// TIA Portal V20 export
FUNCTION_BLOCK "Sequence_1_StackNgBox"   // FB32864, LAD
TITLE = Sequence
// Sequence template programmend in ladder logic
// stored: IsIECCheckEnabled true, MemoryReserve 100, Namespace Unit1.Em12, SetENOAutomatically true
   VAR_INPUT
      unitStatus { ExternalAccessible := 'False'; ExternalVisible := 'False'; ExternalWritable := 'False'} : "LAF_typeUnitStatus";   // Current unit status o be used in this EM
   END_VAR
   VAR
      instSequenceLADControl { ExternalAccessible := 'False'; ExternalVisible := 'False'; ExternalWritable := 'False'} : "LAF_ControlLadSequence";
      instSequenceLADStatus { ExternalAccessible := 'False'; ExternalVisible := 'False'; ExternalWritable := 'False'} : "LAF_StatusLadSequence";
      statTonTime { ExternalAccessible := 'False'; ExternalVisible := 'False'; ExternalWritable := 'False'} : Array[0..9999] of TON_TIME;
      NoDataCheck { S7_SetPoint := 'True'} : "LER_typePartData";
   END_VAR
   VAR_TEMP
      tempCustomerAction : Bool;   // Placeholder for possible actions
      tempDo_nothing_and_wait_for_init : Bool;   // Placeholder for doing nothing
      tempSafeStateCondition : Bool;   // Temp Condition for the equipment module to be in a safe state
   END_VAR
   VAR CONSTANT
      delayTime : Time := T#500ms;
      STEP_IDLE : DInt := 1;
      JOB_1_STEP_01 : DInt := 101;
      JOB_1_STEP_10 : DInt := 110;
      JOB_1_STEP_20 : DInt := 120;
      JOB_1_STEP_30 : DInt := 130;
      JOB_1_STEP_40 : DInt := 140;
      JOB_1_STEP_50 : DInt := 150;
      JOB_1_STEP_60 : DInt := 160;
      JOB_1_STEP_70 : DInt := 170;
      JOB_1_STEP_80 : DInt := 180;
      JOB_1_STEP_90 : DInt := 190;
      JOB_2_STEP_01 : DInt := 201;
      JOB_2_STEP_10 : DInt := 210;
      JOB_2_STEP_20 : DInt := 220;
      JOB_2_STEP_30 : DInt := 230;
      JOB_2_STEP_31 : DInt := 231;
      JOB_2_STEP_40 : DInt := 240;
      JOB_2_STEP_50 : DInt := 250;
      JOB_2_STEP_60 : DInt := 260;
      JOB_2_STEP_70 : DInt := 270;
      JOB_2_STEP_80 : DInt := 280;
      JOB_2_STEP_90 : DInt := 290;
      JOB_3_STEP_01 : DInt := 301;
      JOB_3_STEP_10 : DInt := 310;
      JOB_3_STEP_20 : DInt := 320;
      JOB_3_STEP_30 : DInt := 330;
      JOB_3_STEP_40 : DInt := 340;
      JOB_3_STEP_50 : DInt := 350;
      JOB_3_STEP_60 : DInt := 360;
      JOB_3_STEP_70 : DInt := 370;
      JOB_3_STEP_80 : DInt := 380;
      JOB_3_STEP_90 : DInt := 390;
      STEP_IMMEDIATE_STOP : DInt := 9001;   // Step executed when an immediate stop command is triggered for the sequence (i.e. when unit is in state aborting)
   END_VAR
   VAR_TEMP   // added for the SCL form of the ladder/FBD networks
      _w1 : Bool;
      _w2 : Bool;
   END_VAR
BEGIN

REGION Network 1: BLOCK INFO HEADER
   // (company) / (C) Copyright (year)
   // ---------------------------------------------------------------------------------
   // Title:                             (Title of this block)
   // Comment/Function: (that is implemented in the block)
   // Library/Family:           (that the source is dedicated to)
   // Author:                        (department / person in charge / contact)
   // Target System:          (test system with FW version)
   // Engineering:              TIA Portal (SW version)
   // Restrictions:               (OB types, etc.)
   // Requirements:           (hardware, technological package, etc.)
   // ---------------------------------------------------------------------------------
   // Change log table:
   // Version          | Date             | Signature      | Expert in charge  | Changes applied ------------------------|----------------------|-------------------------|--------------------------------|-----------------------
   // 001.000.000 | yyyy-mm-dd | 0x00000000 | (name of expert) | First released version
END_REGION

REGION Network 2 (SCL): DESCRIPTION
   // This is a template block provided by the Automation Framework. It can be used to create an own project.
   // The Block Info Header is prepared to put in your own data.
   // Description of the block could be added here and the docu created by Code2Docu.
   // 1. Home 동작 시 NG box 감지 유무에 따라 Lock, Unlock이 되면 박스의 위치가 정확하지 않을 때는 불합리하므로 작업자의 수동 작업 필요.
END_REGION

REGION Network 3: ********************* CONTROL *************************
END_REGION

REGION Network 4: Sequence Control ("Enter your Sequins number here")
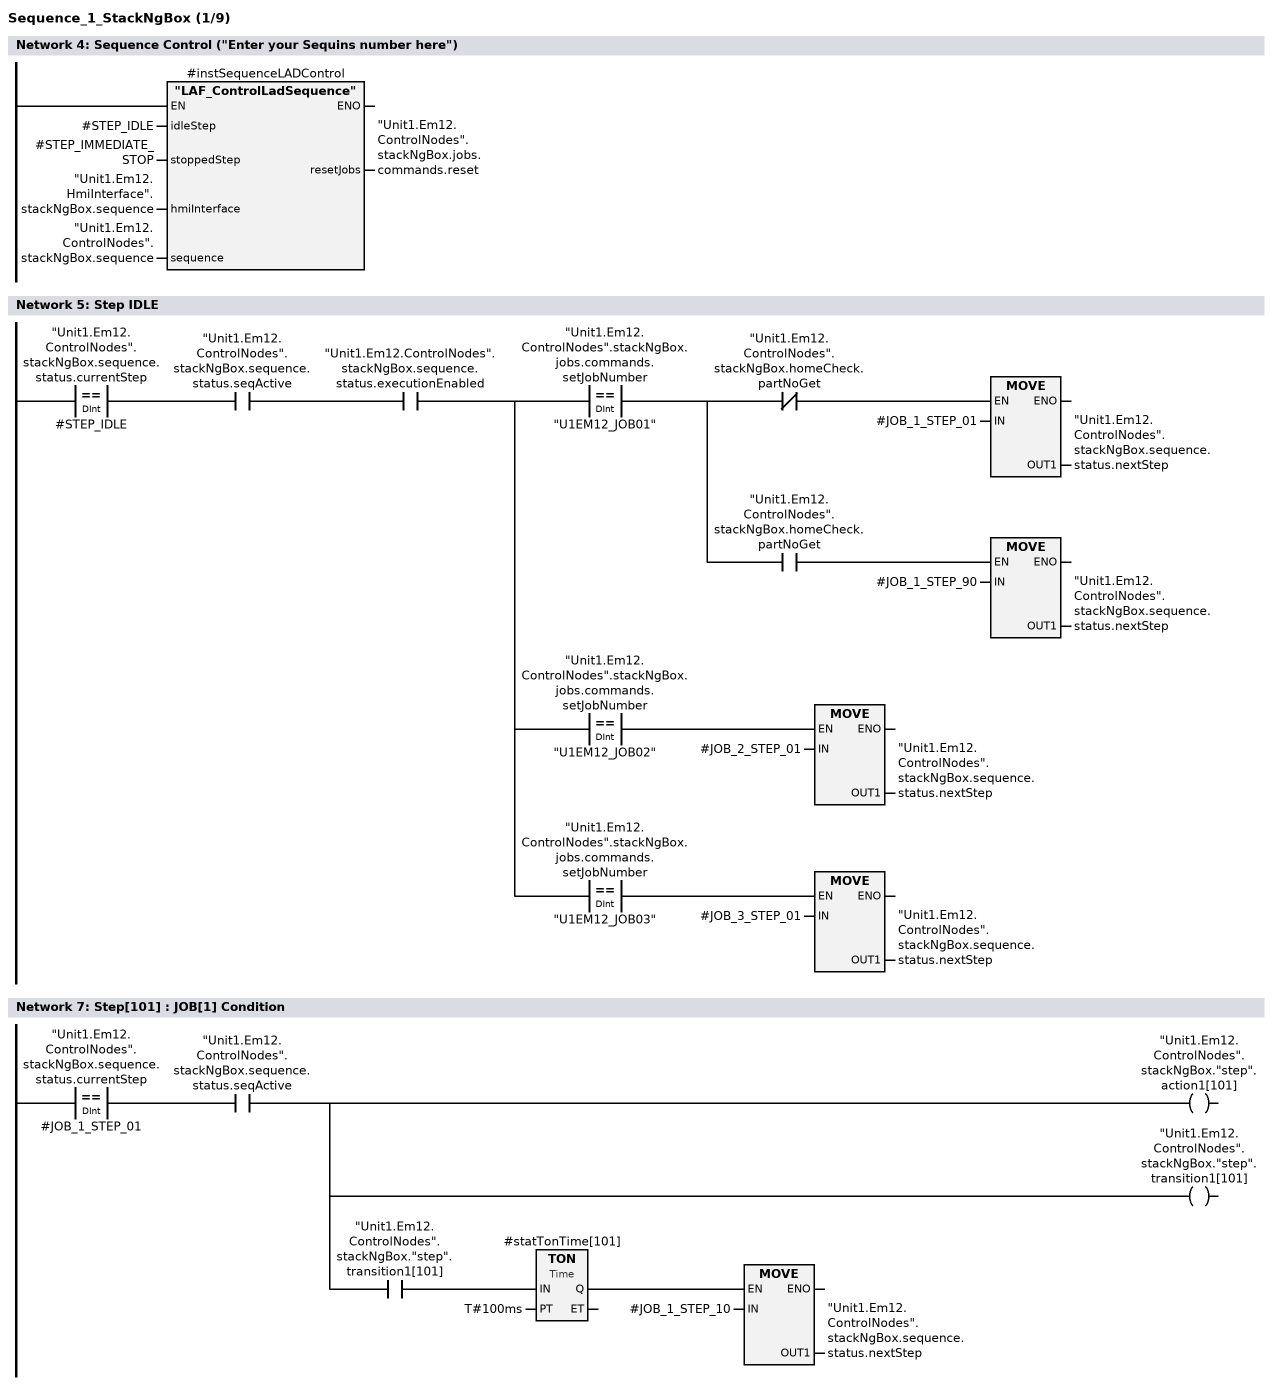
   RUNG wire#powerrail
      #instSequenceLADControl(idleStep := #STEP_IDLE, stoppedStep := #STEP_IMMEDIATE_STOP, hmiInterface := "Unit1.Em12.HmiInterface".stackNgBox.sequence, sequence := "Unit1.Em12.ControlNodes".stackNgBox.sequence, resetJobs => "Unit1.Em12.ControlNodes".stackNgBox.jobs.commands.reset)
   END_RUNG
   // the same network as SCL:
   #instSequenceLADControl(idleStep := #STEP_IDLE,   // "LAF_ControlLadSequence"
                           stoppedStep := #STEP_IMMEDIATE_STOP,
                           hmiInterface := "Unit1.Em12.HmiInterface".stackNgBox.sequence,
                           sequence := "Unit1.Em12.ControlNodes".stackNgBox.sequence,
                           resetJobs => "Unit1.Em12.ControlNodes".stackNgBox.jobs.commands.reset);
END_REGION

REGION Network 5: Step IDLE
   RUNG wire#powerrail
      { S7_Templates := "SrcType := DInt" } EQ_Contact(in1 := "Unit1.Em12.ControlNodes".stackNgBox.sequence.status.currentStep, in2 := #STEP_IDLE)
      Contact( "Unit1.Em12.ControlNodes".stackNgBox.sequence.status.seqActive )
      Contact( "Unit1.Em12.ControlNodes".stackNgBox.sequence.status.executionEnabled )
      wire#w1
      { S7_Templates := "SrcType := DInt" } EQ_Contact(in1 := "Unit1.Em12.ControlNodes".stackNgBox.jobs.commands.setJobNumber, in2 := "U1EM12_JOB01")
      wire#w2
      I_Contact( "Unit1.Em12.ControlNodes".stackNgBox.homeCheck.partNoGet )
      Move(in := #JOB_1_STEP_01, out1 => "Unit1.Em12.ControlNodes".stackNgBox.sequence.status.nextStep)
   END_RUNG
   RUNG wire#w2
      Contact( "Unit1.Em12.ControlNodes".stackNgBox.homeCheck.partNoGet )
      Move(in := #JOB_1_STEP_90, out1 => "Unit1.Em12.ControlNodes".stackNgBox.sequence.status.nextStep)
   END_RUNG
   RUNG wire#w1
      { S7_Templates := "SrcType := DInt" } EQ_Contact(in1 := "Unit1.Em12.ControlNodes".stackNgBox.jobs.commands.setJobNumber, in2 := "U1EM12_JOB02")
      Move(in := #JOB_2_STEP_01, out1 => "Unit1.Em12.ControlNodes".stackNgBox.sequence.status.nextStep)
   END_RUNG
   RUNG wire#w1
      { S7_Templates := "SrcType := DInt" } EQ_Contact(in1 := "Unit1.Em12.ControlNodes".stackNgBox.jobs.commands.setJobNumber, in2 := "U1EM12_JOB03")
      Move(in := #JOB_3_STEP_01, out1 => "Unit1.Em12.ControlNodes".stackNgBox.sequence.status.nextStep)
   END_RUNG
   // the same network as SCL:
   #_w1 := ("Unit1.Em12.ControlNodes".stackNgBox.sequence.status.currentStep = #STEP_IDLE) AND "Unit1.Em12.ControlNodes".stackNgBox.sequence.status.seqActive AND "Unit1.Em12.ControlNodes".stackNgBox.sequence.status.executionEnabled;
   #_w2 := #_w1 AND ("Unit1.Em12.ControlNodes".stackNgBox.jobs.commands.setJobNumber = "U1EM12_JOB01");
   IF #_w2 AND NOT "Unit1.Em12.ControlNodes".stackNgBox.homeCheck.partNoGet THEN
       "Unit1.Em12.ControlNodes".stackNgBox.sequence.status.nextStep := #JOB_1_STEP_01;
   END_IF;
   IF #_w2 AND "Unit1.Em12.ControlNodes".stackNgBox.homeCheck.partNoGet THEN
       "Unit1.Em12.ControlNodes".stackNgBox.sequence.status.nextStep := #JOB_1_STEP_90;
   END_IF;
   IF #_w1 AND ("Unit1.Em12.ControlNodes".stackNgBox.jobs.commands.setJobNumber = "U1EM12_JOB02") THEN
       "Unit1.Em12.ControlNodes".stackNgBox.sequence.status.nextStep := #JOB_2_STEP_01;
   END_IF;
   IF #_w1 AND ("Unit1.Em12.ControlNodes".stackNgBox.jobs.commands.setJobNumber = "U1EM12_JOB03") THEN
       "Unit1.Em12.ControlNodes".stackNgBox.sequence.status.nextStep := #JOB_3_STEP_01;
   END_IF;
END_REGION

REGION Network 6: *************** JOB[1] EM HOMING ************************
END_REGION

REGION Network 7: Step[101] : JOB[1] Condition
   RUNG wire#powerrail
      { S7_Templates := "SrcType := DInt" } EQ_Contact(in1 := "Unit1.Em12.ControlNodes".stackNgBox.sequence.status.currentStep, in2 := #JOB_1_STEP_01)
      Contact( "Unit1.Em12.ControlNodes".stackNgBox.sequence.status.seqActive )
      wire#w1
      Coil( "Unit1.Em12.ControlNodes".stackNgBox."step".action1[101] )
   END_RUNG
   RUNG wire#w1
      Coil( "Unit1.Em12.ControlNodes".stackNgBox."step".transition1[101] )
   END_RUNG
   RUNG wire#w1
      Contact( "Unit1.Em12.ControlNodes".stackNgBox."step".transition1[101] )
      { S7_Templates := "time_type := Time" } #statTonTime[101].TON(pt := T#100ms, et =>)
      Move(in := #JOB_1_STEP_10, out1 => "Unit1.Em12.ControlNodes".stackNgBox.sequence.status.nextStep)
   END_RUNG
   // the same network as SCL:
   "Unit1.Em12.ControlNodes".stackNgBox."step".action1[101] := ("Unit1.Em12.ControlNodes".stackNgBox.sequence.status.currentStep = #JOB_1_STEP_01) AND "Unit1.Em12.ControlNodes".stackNgBox.sequence.status.seqActive;
   "Unit1.Em12.ControlNodes".stackNgBox."step".transition1[101] := ("Unit1.Em12.ControlNodes".stackNgBox.sequence.status.currentStep = #JOB_1_STEP_01) AND "Unit1.Em12.ControlNodes".stackNgBox.sequence.status.seqActive;
   #statTonTime[101].TON(IN := ("Unit1.Em12.ControlNodes".stackNgBox.sequence.status.currentStep = #JOB_1_STEP_01) AND "Unit1.Em12.ControlNodes".stackNgBox.sequence.status.seqActive AND "Unit1.Em12.ControlNodes".stackNgBox."step".transition1[101],
                         PT := T#100ms);
   IF #statTonTime[101].Q THEN
       "Unit1.Em12.ControlNodes".stackNgBox.sequence.status.nextStep := #JOB_1_STEP_10;
   END_IF;
END_REGION

REGION Network 8: Step[110] : Clamp Z Up
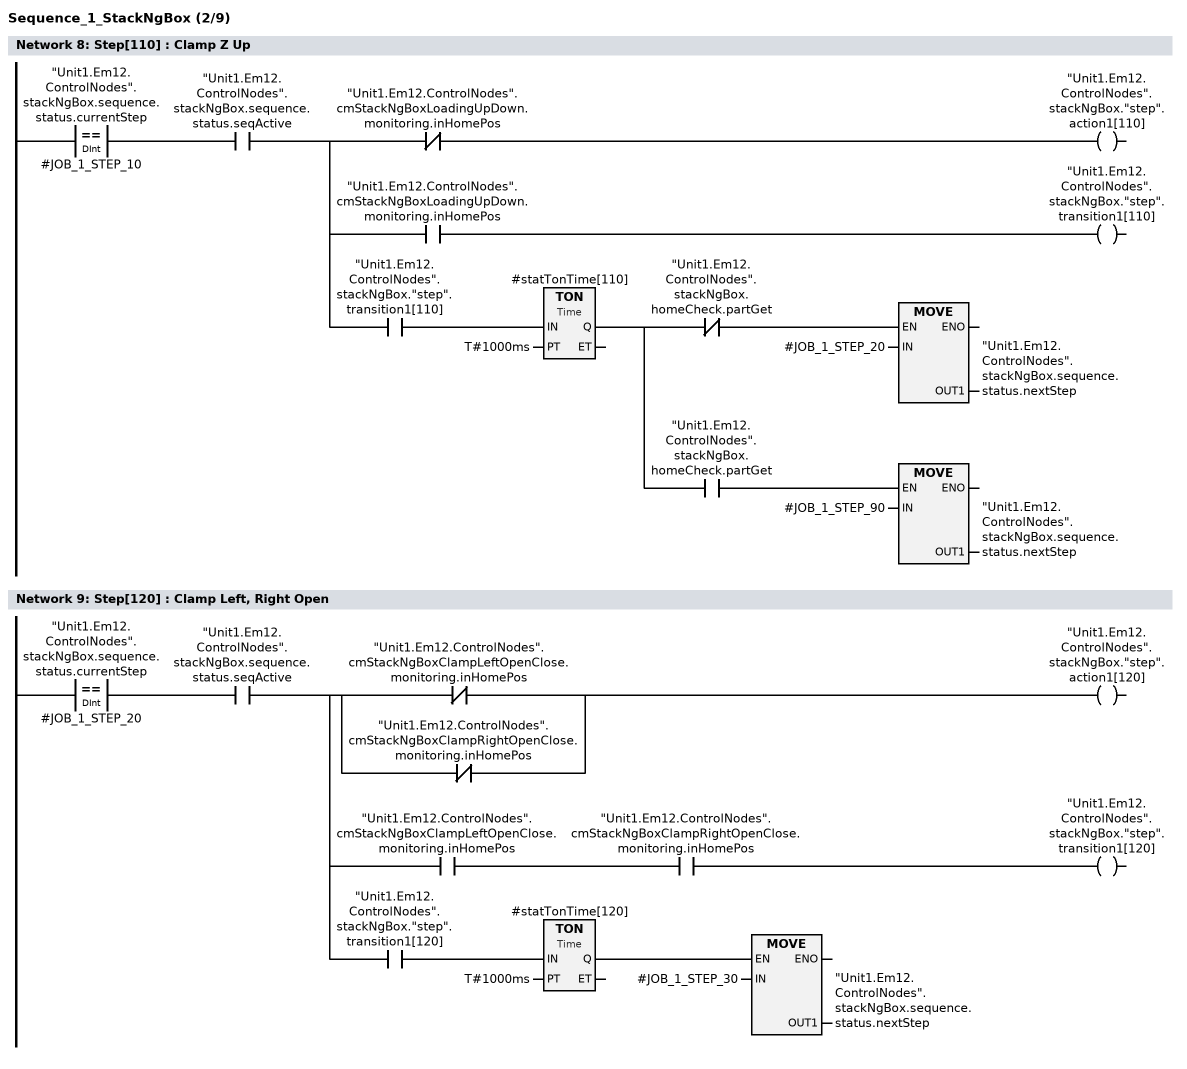
   RUNG wire#powerrail
      { S7_Templates := "SrcType := DInt" } EQ_Contact(in1 := "Unit1.Em12.ControlNodes".stackNgBox.sequence.status.currentStep, in2 := #JOB_1_STEP_10)
      Contact( "Unit1.Em12.ControlNodes".stackNgBox.sequence.status.seqActive )
      wire#w1
      I_Contact( "Unit1.Em12.ControlNodes".cmStackNgBoxLoadingUpDown.monitoring.inHomePos )
      Coil( "Unit1.Em12.ControlNodes".stackNgBox."step".action1[110] )
   END_RUNG
   RUNG wire#w1
      Contact( "Unit1.Em12.ControlNodes".cmStackNgBoxLoadingUpDown.monitoring.inHomePos )
      Coil( "Unit1.Em12.ControlNodes".stackNgBox."step".transition1[110] )
   END_RUNG
   RUNG wire#w1
      Contact( "Unit1.Em12.ControlNodes".stackNgBox."step".transition1[110] )
      { S7_Templates := "time_type := Time" } #statTonTime[110].TON(pt := T#1000ms, et =>)
      wire#w2
      I_Contact( "Unit1.Em12.ControlNodes".stackNgBox.homeCheck.partGet )
      Move(in := #JOB_1_STEP_20, out1 => "Unit1.Em12.ControlNodes".stackNgBox.sequence.status.nextStep)
   END_RUNG
   RUNG wire#w2
      Contact( "Unit1.Em12.ControlNodes".stackNgBox.homeCheck.partGet )
      Move(in := #JOB_1_STEP_90, out1 => "Unit1.Em12.ControlNodes".stackNgBox.sequence.status.nextStep)
   END_RUNG
   // the same network as SCL:
   #_w1 := ("Unit1.Em12.ControlNodes".stackNgBox.sequence.status.currentStep = #JOB_1_STEP_10) AND "Unit1.Em12.ControlNodes".stackNgBox.sequence.status.seqActive;
   "Unit1.Em12.ControlNodes".stackNgBox."step".action1[110] := #_w1 AND NOT "Unit1.Em12.ControlNodes".cmStackNgBoxLoadingUpDown.monitoring.inHomePos;
   "Unit1.Em12.ControlNodes".stackNgBox."step".transition1[110] := #_w1 AND "Unit1.Em12.ControlNodes".cmStackNgBoxLoadingUpDown.monitoring.inHomePos;
   #statTonTime[110].TON(IN := #_w1 AND "Unit1.Em12.ControlNodes".stackNgBox."step".transition1[110],
                         PT := T#1000ms);
   IF #statTonTime[110].Q AND NOT "Unit1.Em12.ControlNodes".stackNgBox.homeCheck.partGet THEN
       "Unit1.Em12.ControlNodes".stackNgBox.sequence.status.nextStep := #JOB_1_STEP_20;
   END_IF;
   IF #statTonTime[110].Q AND "Unit1.Em12.ControlNodes".stackNgBox.homeCheck.partGet THEN
       "Unit1.Em12.ControlNodes".stackNgBox.sequence.status.nextStep := #JOB_1_STEP_90;
   END_IF;
END_REGION

REGION Network 9: Step[120] : Clamp Left, Right Open
   RUNG wire#powerrail
      { S7_Templates := "SrcType := DInt" } EQ_Contact(in1 := "Unit1.Em12.ControlNodes".stackNgBox.sequence.status.currentStep, in2 := #JOB_1_STEP_20)
      Contact( "Unit1.Em12.ControlNodes".stackNgBox.sequence.status.seqActive )
      wire#w1
      I_Contact( "Unit1.Em12.ControlNodes".cmStackNgBoxClampLeftOpenClose.monitoring.inHomePos )
      wire#w2
      Coil( "Unit1.Em12.ControlNodes".stackNgBox."step".action1[120] )
   END_RUNG
   RUNG wire#w1
      I_Contact( "Unit1.Em12.ControlNodes".cmStackNgBoxClampRightOpenClose.monitoring.inHomePos )
   END_RUNG wire#w2
   RUNG wire#w1
      Contact( "Unit1.Em12.ControlNodes".cmStackNgBoxClampLeftOpenClose.monitoring.inHomePos )
      Contact( "Unit1.Em12.ControlNodes".cmStackNgBoxClampRightOpenClose.monitoring.inHomePos )
      Coil( "Unit1.Em12.ControlNodes".stackNgBox."step".transition1[120] )
   END_RUNG
   RUNG wire#w1
      Contact( "Unit1.Em12.ControlNodes".stackNgBox."step".transition1[120] )
      { S7_Templates := "time_type := Time" } #statTonTime[120].TON(pt := T#1000ms, et =>)
      Move(in := #JOB_1_STEP_30, out1 => "Unit1.Em12.ControlNodes".stackNgBox.sequence.status.nextStep)
   END_RUNG
   // the same network as SCL:
   #_w1 := ("Unit1.Em12.ControlNodes".stackNgBox.sequence.status.currentStep = #JOB_1_STEP_20) AND "Unit1.Em12.ControlNodes".stackNgBox.sequence.status.seqActive;
   "Unit1.Em12.ControlNodes".stackNgBox."step".action1[120] := #_w1 AND (NOT "Unit1.Em12.ControlNodes".cmStackNgBoxClampLeftOpenClose.monitoring.inHomePos OR NOT "Unit1.Em12.ControlNodes".cmStackNgBoxClampRightOpenClose.monitoring.inHomePos);
   "Unit1.Em12.ControlNodes".stackNgBox."step".transition1[120] := #_w1 AND "Unit1.Em12.ControlNodes".cmStackNgBoxClampLeftOpenClose.monitoring.inHomePos AND "Unit1.Em12.ControlNodes".cmStackNgBoxClampRightOpenClose.monitoring.inHomePos;
   #statTonTime[120].TON(IN := #_w1 AND "Unit1.Em12.ControlNodes".stackNgBox."step".transition1[120],
                         PT := T#1000ms);
   IF #statTonTime[120].Q THEN
       "Unit1.Em12.ControlNodes".stackNgBox.sequence.status.nextStep := #JOB_1_STEP_30;
   END_IF;
END_REGION

REGION Network 10: Step[130] : Clamp Mover Open
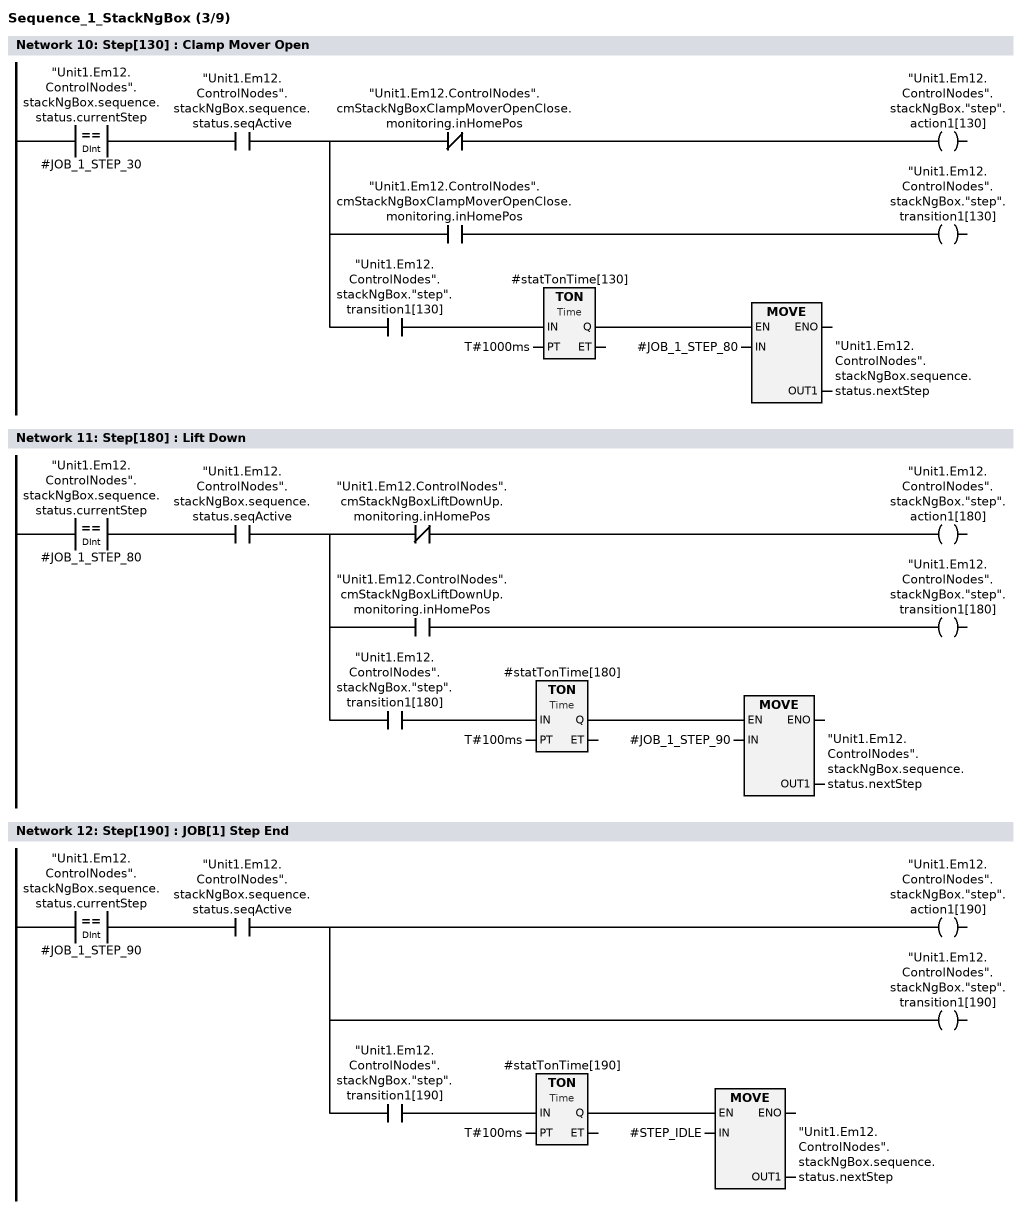
   RUNG wire#powerrail
      { S7_Templates := "SrcType := DInt" } EQ_Contact(in1 := "Unit1.Em12.ControlNodes".stackNgBox.sequence.status.currentStep, in2 := #JOB_1_STEP_30)
      Contact( "Unit1.Em12.ControlNodes".stackNgBox.sequence.status.seqActive )
      wire#w1
      I_Contact( "Unit1.Em12.ControlNodes".cmStackNgBoxClampMoverOpenClose.monitoring.inHomePos )
      Coil( "Unit1.Em12.ControlNodes".stackNgBox."step".action1[130] )
   END_RUNG
   RUNG wire#w1
      Contact( "Unit1.Em12.ControlNodes".cmStackNgBoxClampMoverOpenClose.monitoring.inHomePos )
      Coil( "Unit1.Em12.ControlNodes".stackNgBox."step".transition1[130] )
   END_RUNG
   RUNG wire#w1
      Contact( "Unit1.Em12.ControlNodes".stackNgBox."step".transition1[130] )
      { S7_Templates := "time_type := Time" } #statTonTime[130].TON(pt := T#1000ms, et =>)
      Move(in := #JOB_1_STEP_80, out1 => "Unit1.Em12.ControlNodes".stackNgBox.sequence.status.nextStep)
   END_RUNG
   // the same network as SCL:
   #_w1 := ("Unit1.Em12.ControlNodes".stackNgBox.sequence.status.currentStep = #JOB_1_STEP_30) AND "Unit1.Em12.ControlNodes".stackNgBox.sequence.status.seqActive;
   "Unit1.Em12.ControlNodes".stackNgBox."step".action1[130] := #_w1 AND NOT "Unit1.Em12.ControlNodes".cmStackNgBoxClampMoverOpenClose.monitoring.inHomePos;
   "Unit1.Em12.ControlNodes".stackNgBox."step".transition1[130] := #_w1 AND "Unit1.Em12.ControlNodes".cmStackNgBoxClampMoverOpenClose.monitoring.inHomePos;
   #statTonTime[130].TON(IN := #_w1 AND "Unit1.Em12.ControlNodes".stackNgBox."step".transition1[130],
                         PT := T#1000ms);
   IF #statTonTime[130].Q THEN
       "Unit1.Em12.ControlNodes".stackNgBox.sequence.status.nextStep := #JOB_1_STEP_80;
   END_IF;
END_REGION

REGION Network 11: Step[180] : Lift Down
   RUNG wire#powerrail
      { S7_Templates := "SrcType := DInt" } EQ_Contact(in1 := "Unit1.Em12.ControlNodes".stackNgBox.sequence.status.currentStep, in2 := #JOB_1_STEP_80)
      Contact( "Unit1.Em12.ControlNodes".stackNgBox.sequence.status.seqActive )
      wire#w1
      I_Contact( "Unit1.Em12.ControlNodes".cmStackNgBoxLiftDownUp.monitoring.inHomePos )
      Coil( "Unit1.Em12.ControlNodes".stackNgBox."step".action1[180] )
   END_RUNG
   RUNG wire#w1
      Contact( "Unit1.Em12.ControlNodes".cmStackNgBoxLiftDownUp.monitoring.inHomePos )
      Coil( "Unit1.Em12.ControlNodes".stackNgBox."step".transition1[180] )
   END_RUNG
   RUNG wire#w1
      Contact( "Unit1.Em12.ControlNodes".stackNgBox."step".transition1[180] )
      { S7_Templates := "time_type := Time" } #statTonTime[180].TON(pt := T#100ms, et =>)
      Move(in := #JOB_1_STEP_90, out1 => "Unit1.Em12.ControlNodes".stackNgBox.sequence.status.nextStep)
   END_RUNG
   // the same network as SCL:
   #_w1 := ("Unit1.Em12.ControlNodes".stackNgBox.sequence.status.currentStep = #JOB_1_STEP_80) AND "Unit1.Em12.ControlNodes".stackNgBox.sequence.status.seqActive;
   "Unit1.Em12.ControlNodes".stackNgBox."step".action1[180] := #_w1 AND NOT "Unit1.Em12.ControlNodes".cmStackNgBoxLiftDownUp.monitoring.inHomePos;
   "Unit1.Em12.ControlNodes".stackNgBox."step".transition1[180] := #_w1 AND "Unit1.Em12.ControlNodes".cmStackNgBoxLiftDownUp.monitoring.inHomePos;
   #statTonTime[180].TON(IN := #_w1 AND "Unit1.Em12.ControlNodes".stackNgBox."step".transition1[180],
                         PT := T#100ms);
   IF #statTonTime[180].Q THEN
       "Unit1.Em12.ControlNodes".stackNgBox.sequence.status.nextStep := #JOB_1_STEP_90;
   END_IF;
END_REGION

REGION Network 12: Step[190] : JOB[1] Step End
   RUNG wire#powerrail
      { S7_Templates := "SrcType := DInt" } EQ_Contact(in1 := "Unit1.Em12.ControlNodes".stackNgBox.sequence.status.currentStep, in2 := #JOB_1_STEP_90)
      Contact( "Unit1.Em12.ControlNodes".stackNgBox.sequence.status.seqActive )
      wire#w1
      Coil( "Unit1.Em12.ControlNodes".stackNgBox."step".action1[190] )
   END_RUNG
   RUNG wire#w1
      Coil( "Unit1.Em12.ControlNodes".stackNgBox."step".transition1[190] )
   END_RUNG
   RUNG wire#w1
      Contact( "Unit1.Em12.ControlNodes".stackNgBox."step".transition1[190] )
      { S7_Templates := "time_type := Time" } #statTonTime[190].TON(pt := T#100ms, et =>)
      Move(in := #STEP_IDLE, out1 => "Unit1.Em12.ControlNodes".stackNgBox.sequence.status.nextStep)
   END_RUNG
   // the same network as SCL:
   "Unit1.Em12.ControlNodes".stackNgBox."step".action1[190] := ("Unit1.Em12.ControlNodes".stackNgBox.sequence.status.currentStep = #JOB_1_STEP_90) AND "Unit1.Em12.ControlNodes".stackNgBox.sequence.status.seqActive;
   "Unit1.Em12.ControlNodes".stackNgBox."step".transition1[190] := ("Unit1.Em12.ControlNodes".stackNgBox.sequence.status.currentStep = #JOB_1_STEP_90) AND "Unit1.Em12.ControlNodes".stackNgBox.sequence.status.seqActive;
   #statTonTime[190].TON(IN := ("Unit1.Em12.ControlNodes".stackNgBox.sequence.status.currentStep = #JOB_1_STEP_90) AND "Unit1.Em12.ControlNodes".stackNgBox.sequence.status.seqActive AND "Unit1.Em12.ControlNodes".stackNgBox."step".transition1[190],
                         PT := T#100ms);
   IF #statTonTime[190].Q THEN
       "Unit1.Em12.ControlNodes".stackNgBox.sequence.status.nextStep := #STEP_IDLE;
   END_IF;
END_REGION

REGION Network 13: *************** JOB[2] JR GET=AUTO **********************
END_REGION

REGION Network 14: Step[201] : JOB[2] Condition
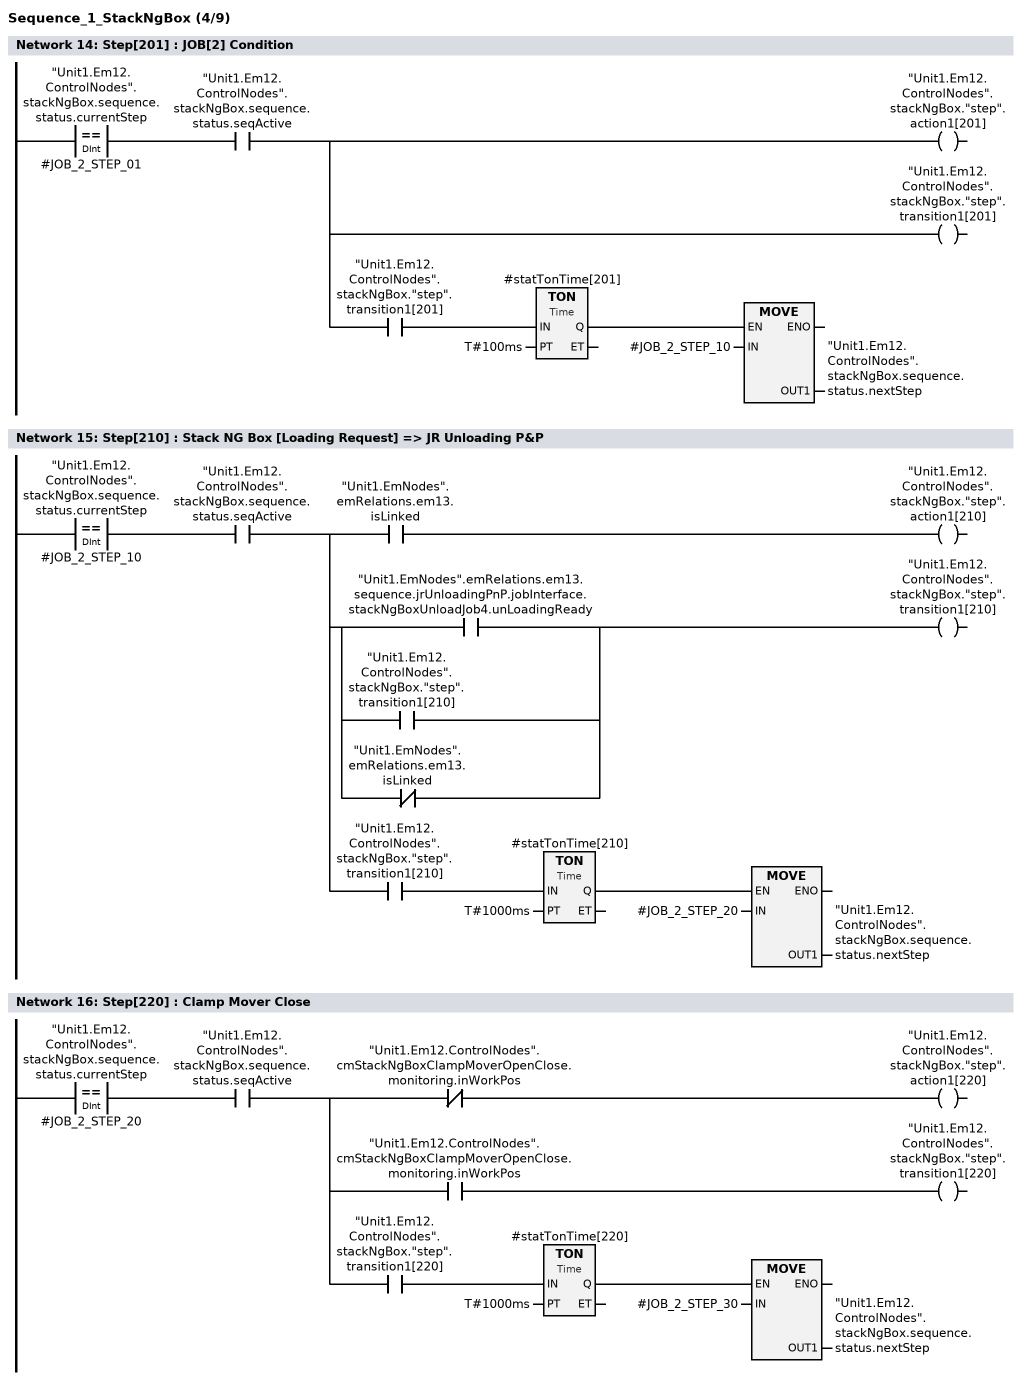
   RUNG wire#powerrail
      { S7_Templates := "SrcType := DInt" } EQ_Contact(in1 := "Unit1.Em12.ControlNodes".stackNgBox.sequence.status.currentStep, in2 := #JOB_2_STEP_01)
      Contact( "Unit1.Em12.ControlNodes".stackNgBox.sequence.status.seqActive )
      wire#w1
      Coil( "Unit1.Em12.ControlNodes".stackNgBox."step".action1[201] )
   END_RUNG
   RUNG wire#w1
      Coil( "Unit1.Em12.ControlNodes".stackNgBox."step".transition1[201] )
   END_RUNG
   RUNG wire#w1
      Contact( "Unit1.Em12.ControlNodes".stackNgBox."step".transition1[201] )
      { S7_Templates := "time_type := Time" } #statTonTime[201].TON(pt := T#100ms, et =>)
      Move(in := #JOB_2_STEP_10, out1 => "Unit1.Em12.ControlNodes".stackNgBox.sequence.status.nextStep)
   END_RUNG
   // the same network as SCL:
   "Unit1.Em12.ControlNodes".stackNgBox."step".action1[201] := ("Unit1.Em12.ControlNodes".stackNgBox.sequence.status.currentStep = #JOB_2_STEP_01) AND "Unit1.Em12.ControlNodes".stackNgBox.sequence.status.seqActive;
   "Unit1.Em12.ControlNodes".stackNgBox."step".transition1[201] := ("Unit1.Em12.ControlNodes".stackNgBox.sequence.status.currentStep = #JOB_2_STEP_01) AND "Unit1.Em12.ControlNodes".stackNgBox.sequence.status.seqActive;
   #statTonTime[201].TON(IN := ("Unit1.Em12.ControlNodes".stackNgBox.sequence.status.currentStep = #JOB_2_STEP_01) AND "Unit1.Em12.ControlNodes".stackNgBox.sequence.status.seqActive AND "Unit1.Em12.ControlNodes".stackNgBox."step".transition1[201],
                         PT := T#100ms);
   IF #statTonTime[201].Q THEN
       "Unit1.Em12.ControlNodes".stackNgBox.sequence.status.nextStep := #JOB_2_STEP_10;
   END_IF;
END_REGION

REGION Network 15: Step[210] : Stack NG Box [Loading Request] => JR Unloading P&P
   RUNG wire#powerrail
      { S7_Templates := "SrcType := DInt" } EQ_Contact(in1 := "Unit1.Em12.ControlNodes".stackNgBox.sequence.status.currentStep, in2 := #JOB_2_STEP_10)
      Contact( "Unit1.Em12.ControlNodes".stackNgBox.sequence.status.seqActive )
      wire#w1
      Contact( "Unit1.EmNodes".emRelations.em13.isLinked )
      Coil( "Unit1.Em12.ControlNodes".stackNgBox."step".action1[210] )
   END_RUNG
   RUNG wire#w1
      Contact( "Unit1.EmNodes".emRelations.em13.sequence.jrUnloadingPnP.jobInterface.stackNgBoxUnloadJob4.unLoadingReady )
      wire#w2
      Coil( "Unit1.Em12.ControlNodes".stackNgBox."step".transition1[210] )
   END_RUNG
   RUNG wire#w1
      Contact( "Unit1.Em12.ControlNodes".stackNgBox."step".transition1[210] )
   END_RUNG wire#w2
   RUNG wire#w1
      I_Contact( "Unit1.EmNodes".emRelations.em13.isLinked )
   END_RUNG wire#w2
   RUNG wire#w1
      Contact( "Unit1.Em12.ControlNodes".stackNgBox."step".transition1[210] )
      { S7_Templates := "time_type := Time" } #statTonTime[210].TON(pt := T#1000ms, et =>)
      Move(in := #JOB_2_STEP_20, out1 => "Unit1.Em12.ControlNodes".stackNgBox.sequence.status.nextStep)
   END_RUNG
   // the same network as SCL:
   #_w1 := ("Unit1.Em12.ControlNodes".stackNgBox.sequence.status.currentStep = #JOB_2_STEP_10) AND "Unit1.Em12.ControlNodes".stackNgBox.sequence.status.seqActive;
   "Unit1.Em12.ControlNodes".stackNgBox."step".action1[210] := #_w1 AND "Unit1.EmNodes".emRelations.em13.isLinked;
   "Unit1.Em12.ControlNodes".stackNgBox."step".transition1[210] := #_w1 AND ("Unit1.EmNodes".emRelations.em13.sequence.jrUnloadingPnP.jobInterface.stackNgBoxUnloadJob4.unLoadingReady OR "Unit1.Em12.ControlNodes".stackNgBox."step".transition1[210] OR NOT "Unit1.EmNodes".emRelations.em13.isLinked);
   #statTonTime[210].TON(IN := #_w1 AND "Unit1.Em12.ControlNodes".stackNgBox."step".transition1[210],
                         PT := T#1000ms);
   IF #statTonTime[210].Q THEN
       "Unit1.Em12.ControlNodes".stackNgBox.sequence.status.nextStep := #JOB_2_STEP_20;
   END_IF;
END_REGION

REGION Network 16: Step[220] : Clamp Mover Close
   RUNG wire#powerrail
      { S7_Templates := "SrcType := DInt" } EQ_Contact(in1 := "Unit1.Em12.ControlNodes".stackNgBox.sequence.status.currentStep, in2 := #JOB_2_STEP_20)
      Contact( "Unit1.Em12.ControlNodes".stackNgBox.sequence.status.seqActive )
      wire#w1
      I_Contact( "Unit1.Em12.ControlNodes".cmStackNgBoxClampMoverOpenClose.monitoring.inWorkPos )
      Coil( "Unit1.Em12.ControlNodes".stackNgBox."step".action1[220] )
   END_RUNG
   RUNG wire#w1
      Contact( "Unit1.Em12.ControlNodes".cmStackNgBoxClampMoverOpenClose.monitoring.inWorkPos )
      Coil( "Unit1.Em12.ControlNodes".stackNgBox."step".transition1[220] )
   END_RUNG
   RUNG wire#w1
      Contact( "Unit1.Em12.ControlNodes".stackNgBox."step".transition1[220] )
      { S7_Templates := "time_type := Time" } #statTonTime[220].TON(pt := T#1000ms, et =>)
      Move(in := #JOB_2_STEP_30, out1 => "Unit1.Em12.ControlNodes".stackNgBox.sequence.status.nextStep)
   END_RUNG
   // the same network as SCL:
   #_w1 := ("Unit1.Em12.ControlNodes".stackNgBox.sequence.status.currentStep = #JOB_2_STEP_20) AND "Unit1.Em12.ControlNodes".stackNgBox.sequence.status.seqActive;
   "Unit1.Em12.ControlNodes".stackNgBox."step".action1[220] := #_w1 AND NOT "Unit1.Em12.ControlNodes".cmStackNgBoxClampMoverOpenClose.monitoring.inWorkPos;
   "Unit1.Em12.ControlNodes".stackNgBox."step".transition1[220] := #_w1 AND "Unit1.Em12.ControlNodes".cmStackNgBoxClampMoverOpenClose.monitoring.inWorkPos;
   #statTonTime[220].TON(IN := #_w1 AND "Unit1.Em12.ControlNodes".stackNgBox."step".transition1[220],
                         PT := T#1000ms);
   IF #statTonTime[220].Q THEN
       "Unit1.Em12.ControlNodes".stackNgBox.sequence.status.nextStep := #JOB_2_STEP_30;
   END_IF;
END_REGION

REGION Network 17: Step[230] : Clamp Left, Right Close
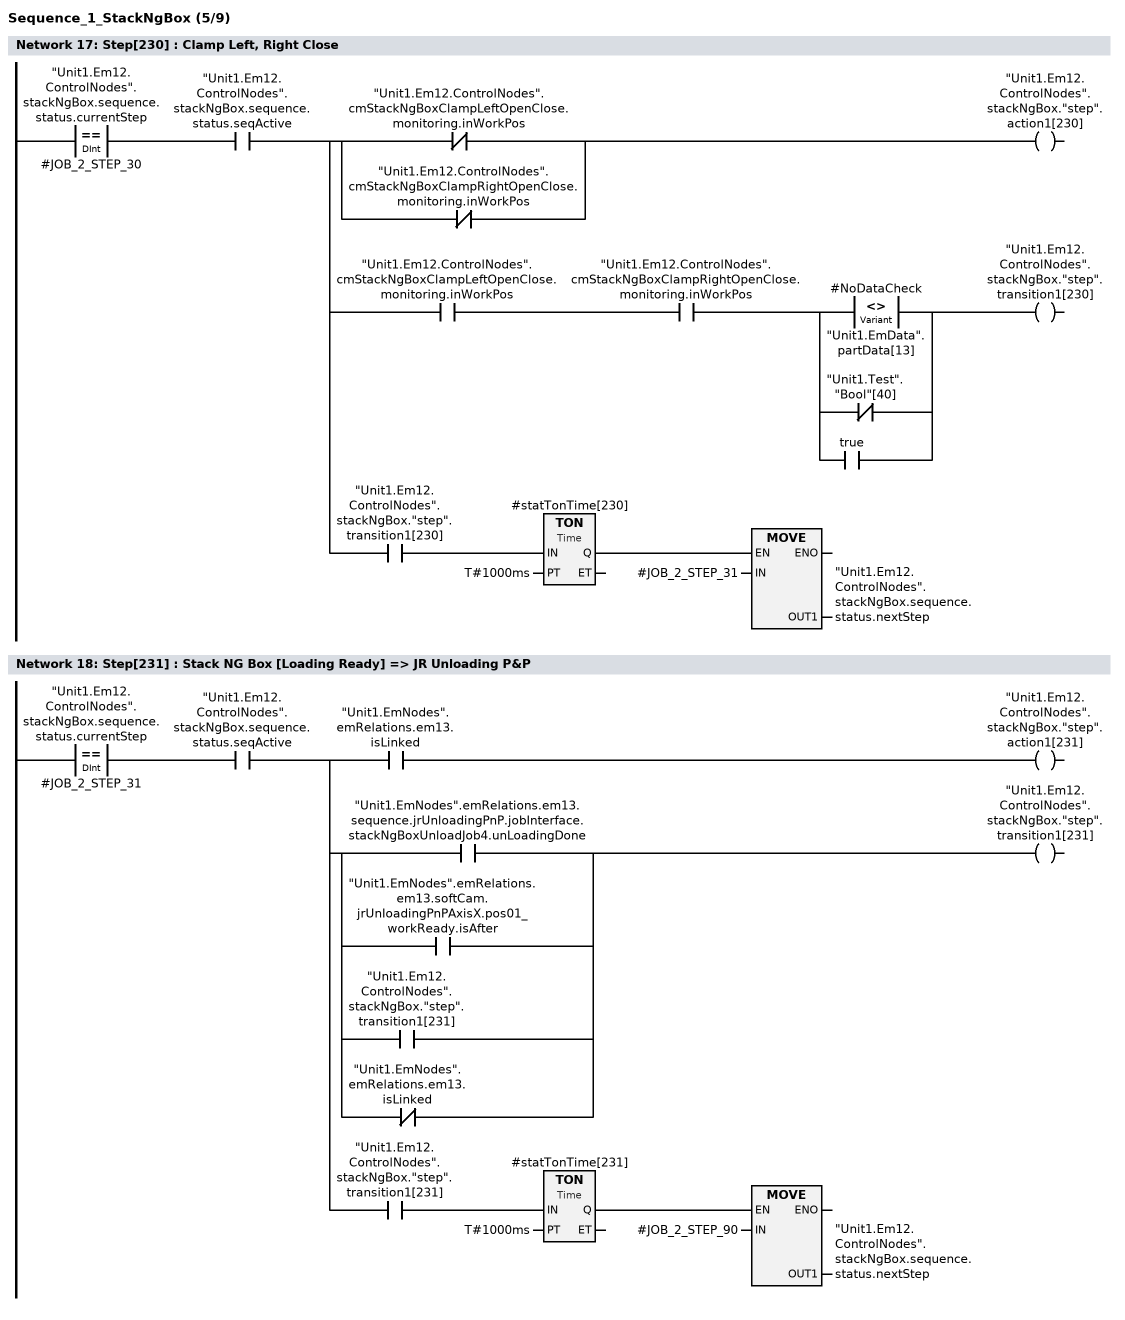
   RUNG wire#powerrail
      { S7_Templates := "SrcType := DInt" } EQ_Contact(in1 := "Unit1.Em12.ControlNodes".stackNgBox.sequence.status.currentStep, in2 := #JOB_2_STEP_30)
      Contact( "Unit1.Em12.ControlNodes".stackNgBox.sequence.status.seqActive )
      wire#w1
      I_Contact( "Unit1.Em12.ControlNodes".cmStackNgBoxClampLeftOpenClose.monitoring.inWorkPos )
      wire#w2
      Coil( "Unit1.Em12.ControlNodes".stackNgBox."step".action1[230] )
   END_RUNG
   RUNG wire#w1
      I_Contact( "Unit1.Em12.ControlNodes".cmStackNgBoxClampRightOpenClose.monitoring.inWorkPos )
   END_RUNG wire#w2
   RUNG wire#w1
      Contact( "Unit1.Em12.ControlNodes".cmStackNgBoxClampLeftOpenClose.monitoring.inWorkPos )
      Contact( "Unit1.Em12.ControlNodes".cmStackNgBoxClampRightOpenClose.monitoring.inWorkPos )
      wire#w3
      { S7_Templates := "SrcType := Variant" } NE_Contact(in1 := #NoDataCheck, in2 := "Unit1.EmData".partData[13])
      wire#w4
      Coil( "Unit1.Em12.ControlNodes".stackNgBox."step".transition1[230] )
   END_RUNG
   RUNG wire#w3
      I_Contact( "Unit1.Test"."Bool"[40] )
   END_RUNG wire#w4
   RUNG wire#w3
      Contact( true )
   END_RUNG wire#w4
   RUNG wire#w1
      Contact( "Unit1.Em12.ControlNodes".stackNgBox."step".transition1[230] )
      { S7_Templates := "time_type := Time" } #statTonTime[230].TON(pt := T#1000ms, et =>)
      Move(in := #JOB_2_STEP_31, out1 => "Unit1.Em12.ControlNodes".stackNgBox.sequence.status.nextStep)
   END_RUNG
   // the same network as SCL:
   #_w1 := ("Unit1.Em12.ControlNodes".stackNgBox.sequence.status.currentStep = #JOB_2_STEP_30) AND "Unit1.Em12.ControlNodes".stackNgBox.sequence.status.seqActive;
   "Unit1.Em12.ControlNodes".stackNgBox."step".action1[230] := #_w1 AND (NOT "Unit1.Em12.ControlNodes".cmStackNgBoxClampLeftOpenClose.monitoring.inWorkPos OR NOT "Unit1.Em12.ControlNodes".cmStackNgBoxClampRightOpenClose.monitoring.inWorkPos);
   "Unit1.Em12.ControlNodes".stackNgBox."step".transition1[230] := #_w1 AND "Unit1.Em12.ControlNodes".cmStackNgBoxClampLeftOpenClose.monitoring.inWorkPos AND "Unit1.Em12.ControlNodes".cmStackNgBoxClampRightOpenClose.monitoring.inWorkPos AND ((#NoDataCheck <> "Unit1.EmData".partData[13]) OR NOT "Unit1.Test"."Bool"[40] OR true);
   #statTonTime[230].TON(IN := #_w1 AND "Unit1.Em12.ControlNodes".stackNgBox."step".transition1[230],
                         PT := T#1000ms);
   IF #statTonTime[230].Q THEN
       "Unit1.Em12.ControlNodes".stackNgBox.sequence.status.nextStep := #JOB_2_STEP_31;
   END_IF;
END_REGION

REGION Network 18: Step[231] : Stack NG Box [Loading Ready] => JR Unloading P&P
   RUNG wire#powerrail
      { S7_Templates := "SrcType := DInt" } EQ_Contact(in1 := "Unit1.Em12.ControlNodes".stackNgBox.sequence.status.currentStep, in2 := #JOB_2_STEP_31)
      Contact( "Unit1.Em12.ControlNodes".stackNgBox.sequence.status.seqActive )
      wire#w1
      Contact( "Unit1.EmNodes".emRelations.em13.isLinked )
      Coil( "Unit1.Em12.ControlNodes".stackNgBox."step".action1[231] )
   END_RUNG
   RUNG wire#w1
      Contact( "Unit1.EmNodes".emRelations.em13.sequence.jrUnloadingPnP.jobInterface.stackNgBoxUnloadJob4.unLoadingDone )
      wire#w2
      Coil( "Unit1.Em12.ControlNodes".stackNgBox."step".transition1[231] )
   END_RUNG
   RUNG wire#w1
      Contact( "Unit1.EmNodes".emRelations.em13.softCam.jrUnIoadingPnPAxisX.pos01_workReady.isAfter )
   END_RUNG wire#w2
   RUNG wire#w1
      Contact( "Unit1.Em12.ControlNodes".stackNgBox."step".transition1[231] )
   END_RUNG wire#w2
   RUNG wire#w1
      I_Contact( "Unit1.EmNodes".emRelations.em13.isLinked )
   END_RUNG wire#w2
   RUNG wire#w1
      Contact( "Unit1.Em12.ControlNodes".stackNgBox."step".transition1[231] )
      { S7_Templates := "time_type := Time" } #statTonTime[231].TON(pt := T#1000ms, et =>)
      Move(in := #JOB_2_STEP_90, out1 => "Unit1.Em12.ControlNodes".stackNgBox.sequence.status.nextStep)
   END_RUNG
   // the same network as SCL:
   #_w1 := ("Unit1.Em12.ControlNodes".stackNgBox.sequence.status.currentStep = #JOB_2_STEP_31) AND "Unit1.Em12.ControlNodes".stackNgBox.sequence.status.seqActive;
   "Unit1.Em12.ControlNodes".stackNgBox."step".action1[231] := #_w1 AND "Unit1.EmNodes".emRelations.em13.isLinked;
   "Unit1.Em12.ControlNodes".stackNgBox."step".transition1[231] := #_w1 AND ("Unit1.EmNodes".emRelations.em13.sequence.jrUnloadingPnP.jobInterface.stackNgBoxUnloadJob4.unLoadingDone OR "Unit1.EmNodes".emRelations.em13.softCam.jrUnIoadingPnPAxisX.pos01_workReady.isAfter OR "Unit1.Em12.ControlNodes".stackNgBox."step".transition1[231] OR NOT "Unit1.EmNodes".emRelations.em13.isLinked);
   #statTonTime[231].TON(IN := #_w1 AND "Unit1.Em12.ControlNodes".stackNgBox."step".transition1[231],
                         PT := T#1000ms);
   IF #statTonTime[231].Q THEN
       "Unit1.Em12.ControlNodes".stackNgBox.sequence.status.nextStep := #JOB_2_STEP_90;
   END_IF;
END_REGION

REGION Network 19: Step[290] : JOB[2] Step End
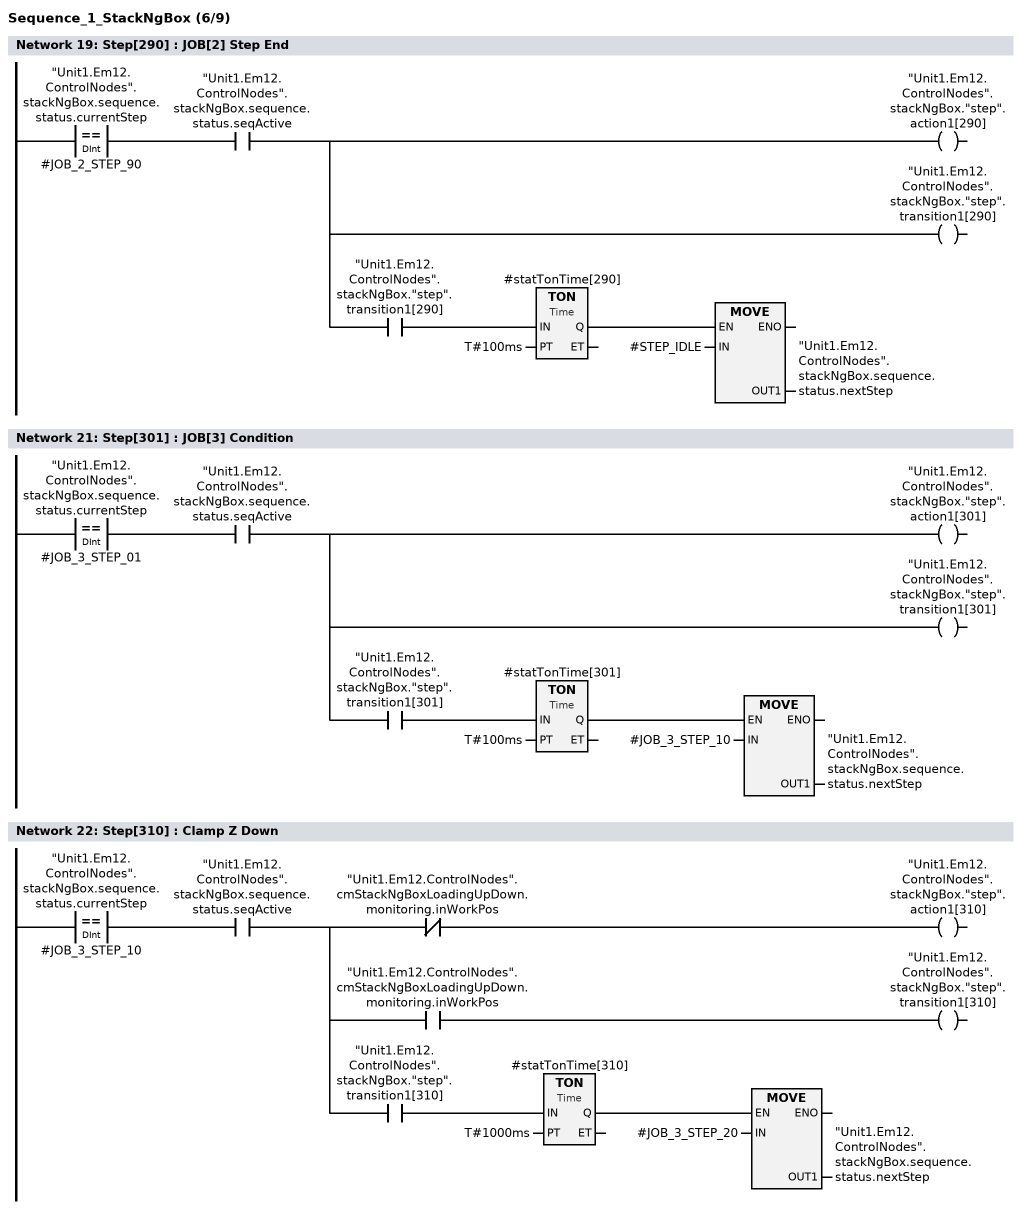
   RUNG wire#powerrail
      { S7_Templates := "SrcType := DInt" } EQ_Contact(in1 := "Unit1.Em12.ControlNodes".stackNgBox.sequence.status.currentStep, in2 := #JOB_2_STEP_90)
      Contact( "Unit1.Em12.ControlNodes".stackNgBox.sequence.status.seqActive )
      wire#w1
      Coil( "Unit1.Em12.ControlNodes".stackNgBox."step".action1[290] )
   END_RUNG
   RUNG wire#w1
      Coil( "Unit1.Em12.ControlNodes".stackNgBox."step".transition1[290] )
   END_RUNG
   RUNG wire#w1
      Contact( "Unit1.Em12.ControlNodes".stackNgBox."step".transition1[290] )
      { S7_Templates := "time_type := Time" } #statTonTime[290].TON(pt := T#100ms, et =>)
      Move(in := #STEP_IDLE, out1 => "Unit1.Em12.ControlNodes".stackNgBox.sequence.status.nextStep)
   END_RUNG
   // the same network as SCL:
   "Unit1.Em12.ControlNodes".stackNgBox."step".action1[290] := ("Unit1.Em12.ControlNodes".stackNgBox.sequence.status.currentStep = #JOB_2_STEP_90) AND "Unit1.Em12.ControlNodes".stackNgBox.sequence.status.seqActive;
   "Unit1.Em12.ControlNodes".stackNgBox."step".transition1[290] := ("Unit1.Em12.ControlNodes".stackNgBox.sequence.status.currentStep = #JOB_2_STEP_90) AND "Unit1.Em12.ControlNodes".stackNgBox.sequence.status.seqActive;
   #statTonTime[290].TON(IN := ("Unit1.Em12.ControlNodes".stackNgBox.sequence.status.currentStep = #JOB_2_STEP_90) AND "Unit1.Em12.ControlNodes".stackNgBox.sequence.status.seqActive AND "Unit1.Em12.ControlNodes".stackNgBox."step".transition1[290],
                         PT := T#100ms);
   IF #statTonTime[290].Q THEN
       "Unit1.Em12.ControlNodes".stackNgBox.sequence.status.nextStep := #STEP_IDLE;
   END_IF;
END_REGION

REGION Network 20: **************** JOB[3] JR PUT=AUTO **********************
END_REGION

REGION Network 21: Step[301] : JOB[3] Condition
   RUNG wire#powerrail
      { S7_Templates := "SrcType := DInt" } EQ_Contact(in1 := "Unit1.Em12.ControlNodes".stackNgBox.sequence.status.currentStep, in2 := #JOB_3_STEP_01)
      Contact( "Unit1.Em12.ControlNodes".stackNgBox.sequence.status.seqActive )
      wire#w1
      Coil( "Unit1.Em12.ControlNodes".stackNgBox."step".action1[301] )
   END_RUNG
   RUNG wire#w1
      Coil( "Unit1.Em12.ControlNodes".stackNgBox."step".transition1[301] )
   END_RUNG
   RUNG wire#w1
      Contact( "Unit1.Em12.ControlNodes".stackNgBox."step".transition1[301] )
      { S7_Templates := "time_type := Time" } #statTonTime[301].TON(pt := T#100ms, et =>)
      Move(in := #JOB_3_STEP_10, out1 => "Unit1.Em12.ControlNodes".stackNgBox.sequence.status.nextStep)
   END_RUNG
   // the same network as SCL:
   "Unit1.Em12.ControlNodes".stackNgBox."step".action1[301] := ("Unit1.Em12.ControlNodes".stackNgBox.sequence.status.currentStep = #JOB_3_STEP_01) AND "Unit1.Em12.ControlNodes".stackNgBox.sequence.status.seqActive;
   "Unit1.Em12.ControlNodes".stackNgBox."step".transition1[301] := ("Unit1.Em12.ControlNodes".stackNgBox.sequence.status.currentStep = #JOB_3_STEP_01) AND "Unit1.Em12.ControlNodes".stackNgBox.sequence.status.seqActive;
   #statTonTime[301].TON(IN := ("Unit1.Em12.ControlNodes".stackNgBox.sequence.status.currentStep = #JOB_3_STEP_01) AND "Unit1.Em12.ControlNodes".stackNgBox.sequence.status.seqActive AND "Unit1.Em12.ControlNodes".stackNgBox."step".transition1[301],
                         PT := T#100ms);
   IF #statTonTime[301].Q THEN
       "Unit1.Em12.ControlNodes".stackNgBox.sequence.status.nextStep := #JOB_3_STEP_10;
   END_IF;
END_REGION

REGION Network 22: Step[310] : Clamp Z Down
   RUNG wire#powerrail
      { S7_Templates := "SrcType := DInt" } EQ_Contact(in1 := "Unit1.Em12.ControlNodes".stackNgBox.sequence.status.currentStep, in2 := #JOB_3_STEP_10)
      Contact( "Unit1.Em12.ControlNodes".stackNgBox.sequence.status.seqActive )
      wire#w1
      I_Contact( "Unit1.Em12.ControlNodes".cmStackNgBoxLoadingUpDown.monitoring.inWorkPos )
      Coil( "Unit1.Em12.ControlNodes".stackNgBox."step".action1[310] )
   END_RUNG
   RUNG wire#w1
      Contact( "Unit1.Em12.ControlNodes".cmStackNgBoxLoadingUpDown.monitoring.inWorkPos )
      Coil( "Unit1.Em12.ControlNodes".stackNgBox."step".transition1[310] )
   END_RUNG
   RUNG wire#w1
      Contact( "Unit1.Em12.ControlNodes".stackNgBox."step".transition1[310] )
      { S7_Templates := "time_type := Time" } #statTonTime[310].TON(pt := T#1000ms, et =>)
      Move(in := #JOB_3_STEP_20, out1 => "Unit1.Em12.ControlNodes".stackNgBox.sequence.status.nextStep)
   END_RUNG
   // the same network as SCL:
   #_w1 := ("Unit1.Em12.ControlNodes".stackNgBox.sequence.status.currentStep = #JOB_3_STEP_10) AND "Unit1.Em12.ControlNodes".stackNgBox.sequence.status.seqActive;
   "Unit1.Em12.ControlNodes".stackNgBox."step".action1[310] := #_w1 AND NOT "Unit1.Em12.ControlNodes".cmStackNgBoxLoadingUpDown.monitoring.inWorkPos;
   "Unit1.Em12.ControlNodes".stackNgBox."step".transition1[310] := #_w1 AND "Unit1.Em12.ControlNodes".cmStackNgBoxLoadingUpDown.monitoring.inWorkPos;
   #statTonTime[310].TON(IN := #_w1 AND "Unit1.Em12.ControlNodes".stackNgBox."step".transition1[310],
                         PT := T#1000ms);
   IF #statTonTime[310].Q THEN
       "Unit1.Em12.ControlNodes".stackNgBox.sequence.status.nextStep := #JOB_3_STEP_20;
   END_IF;
END_REGION

REGION Network 23: Step[320] : Clamp Left, Right Open
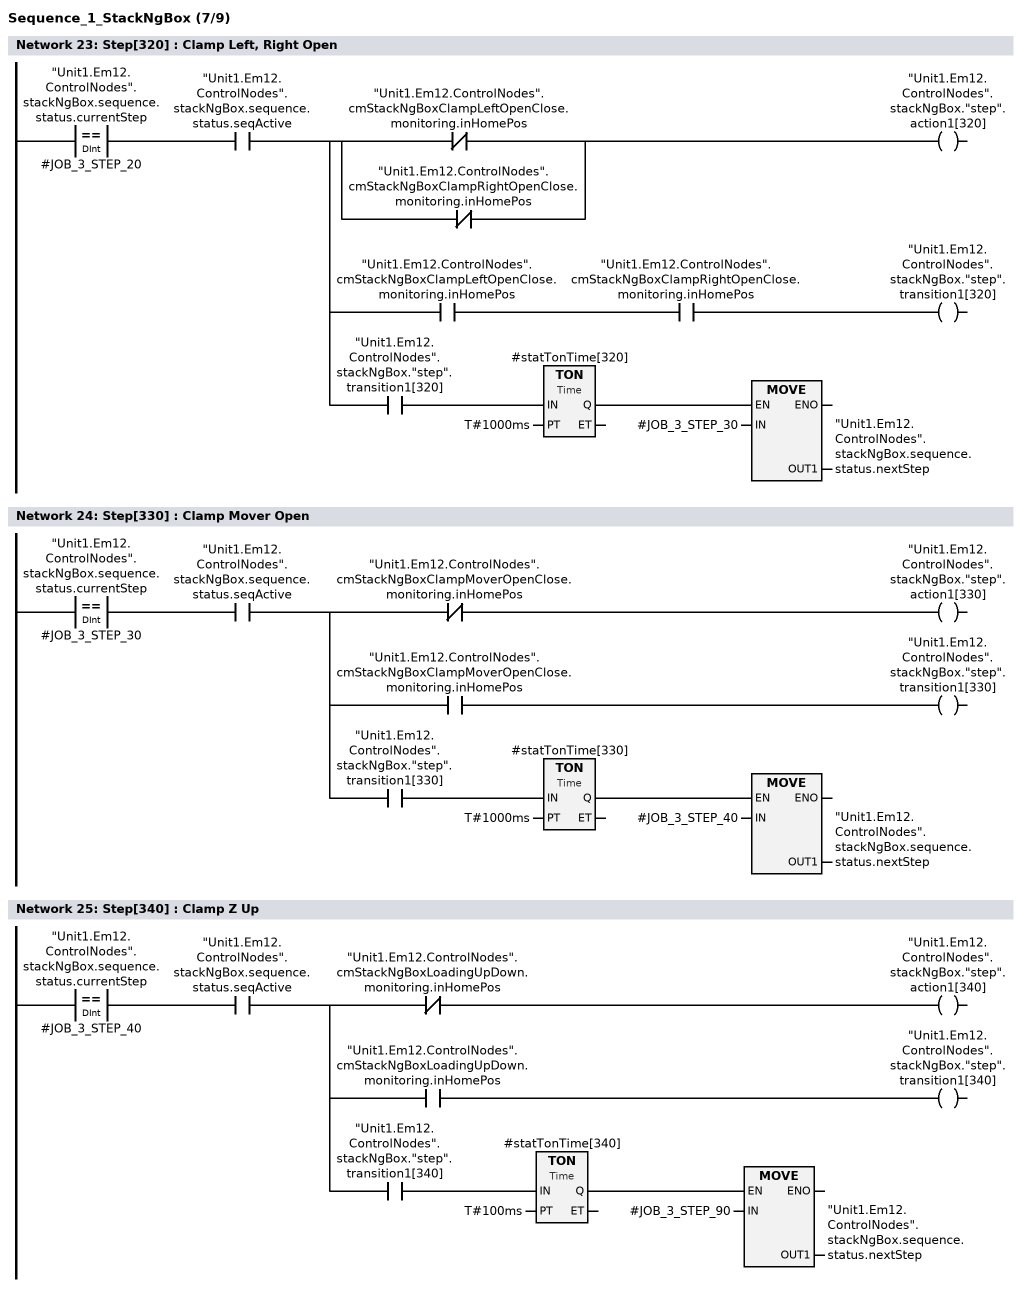
   RUNG wire#powerrail
      { S7_Templates := "SrcType := DInt" } EQ_Contact(in1 := "Unit1.Em12.ControlNodes".stackNgBox.sequence.status.currentStep, in2 := #JOB_3_STEP_20)
      Contact( "Unit1.Em12.ControlNodes".stackNgBox.sequence.status.seqActive )
      wire#w1
      I_Contact( "Unit1.Em12.ControlNodes".cmStackNgBoxClampLeftOpenClose.monitoring.inHomePos )
      wire#w2
      Coil( "Unit1.Em12.ControlNodes".stackNgBox."step".action1[320] )
   END_RUNG
   RUNG wire#w1
      I_Contact( "Unit1.Em12.ControlNodes".cmStackNgBoxClampRightOpenClose.monitoring.inHomePos )
   END_RUNG wire#w2
   RUNG wire#w1
      Contact( "Unit1.Em12.ControlNodes".cmStackNgBoxClampLeftOpenClose.monitoring.inHomePos )
      Contact( "Unit1.Em12.ControlNodes".cmStackNgBoxClampRightOpenClose.monitoring.inHomePos )
      Coil( "Unit1.Em12.ControlNodes".stackNgBox."step".transition1[320] )
   END_RUNG
   RUNG wire#w1
      Contact( "Unit1.Em12.ControlNodes".stackNgBox."step".transition1[320] )
      { S7_Templates := "time_type := Time" } #statTonTime[320].TON(pt := T#1000ms, et =>)
      Move(in := #JOB_3_STEP_30, out1 => "Unit1.Em12.ControlNodes".stackNgBox.sequence.status.nextStep)
   END_RUNG
   // the same network as SCL:
   #_w1 := ("Unit1.Em12.ControlNodes".stackNgBox.sequence.status.currentStep = #JOB_3_STEP_20) AND "Unit1.Em12.ControlNodes".stackNgBox.sequence.status.seqActive;
   "Unit1.Em12.ControlNodes".stackNgBox."step".action1[320] := #_w1 AND (NOT "Unit1.Em12.ControlNodes".cmStackNgBoxClampLeftOpenClose.monitoring.inHomePos OR NOT "Unit1.Em12.ControlNodes".cmStackNgBoxClampRightOpenClose.monitoring.inHomePos);
   "Unit1.Em12.ControlNodes".stackNgBox."step".transition1[320] := #_w1 AND "Unit1.Em12.ControlNodes".cmStackNgBoxClampLeftOpenClose.monitoring.inHomePos AND "Unit1.Em12.ControlNodes".cmStackNgBoxClampRightOpenClose.monitoring.inHomePos;
   #statTonTime[320].TON(IN := #_w1 AND "Unit1.Em12.ControlNodes".stackNgBox."step".transition1[320],
                         PT := T#1000ms);
   IF #statTonTime[320].Q THEN
       "Unit1.Em12.ControlNodes".stackNgBox.sequence.status.nextStep := #JOB_3_STEP_30;
   END_IF;
END_REGION

REGION Network 24: Step[330] : Clamp Mover Open
   RUNG wire#powerrail
      { S7_Templates := "SrcType := DInt" } EQ_Contact(in1 := "Unit1.Em12.ControlNodes".stackNgBox.sequence.status.currentStep, in2 := #JOB_3_STEP_30)
      Contact( "Unit1.Em12.ControlNodes".stackNgBox.sequence.status.seqActive )
      wire#w1
      I_Contact( "Unit1.Em12.ControlNodes".cmStackNgBoxClampMoverOpenClose.monitoring.inHomePos )
      Coil( "Unit1.Em12.ControlNodes".stackNgBox."step".action1[330] )
   END_RUNG
   RUNG wire#w1
      Contact( "Unit1.Em12.ControlNodes".cmStackNgBoxClampMoverOpenClose.monitoring.inHomePos )
      Coil( "Unit1.Em12.ControlNodes".stackNgBox."step".transition1[330] )
   END_RUNG
   RUNG wire#w1
      Contact( "Unit1.Em12.ControlNodes".stackNgBox."step".transition1[330] )
      { S7_Templates := "time_type := Time" } #statTonTime[330].TON(pt := T#1000ms, et =>)
      Move(in := #JOB_3_STEP_40, out1 => "Unit1.Em12.ControlNodes".stackNgBox.sequence.status.nextStep)
   END_RUNG
   // the same network as SCL:
   #_w1 := ("Unit1.Em12.ControlNodes".stackNgBox.sequence.status.currentStep = #JOB_3_STEP_30) AND "Unit1.Em12.ControlNodes".stackNgBox.sequence.status.seqActive;
   "Unit1.Em12.ControlNodes".stackNgBox."step".action1[330] := #_w1 AND NOT "Unit1.Em12.ControlNodes".cmStackNgBoxClampMoverOpenClose.monitoring.inHomePos;
   "Unit1.Em12.ControlNodes".stackNgBox."step".transition1[330] := #_w1 AND "Unit1.Em12.ControlNodes".cmStackNgBoxClampMoverOpenClose.monitoring.inHomePos;
   #statTonTime[330].TON(IN := #_w1 AND "Unit1.Em12.ControlNodes".stackNgBox."step".transition1[330],
                         PT := T#1000ms);
   IF #statTonTime[330].Q THEN
       "Unit1.Em12.ControlNodes".stackNgBox.sequence.status.nextStep := #JOB_3_STEP_40;
   END_IF;
END_REGION

REGION Network 25: Step[340] : Clamp Z Up
   RUNG wire#powerrail
      { S7_Templates := "SrcType := DInt" } EQ_Contact(in1 := "Unit1.Em12.ControlNodes".stackNgBox.sequence.status.currentStep, in2 := #JOB_3_STEP_40)
      Contact( "Unit1.Em12.ControlNodes".stackNgBox.sequence.status.seqActive )
      wire#w1
      I_Contact( "Unit1.Em12.ControlNodes".cmStackNgBoxLoadingUpDown.monitoring.inHomePos )
      Coil( "Unit1.Em12.ControlNodes".stackNgBox."step".action1[340] )
   END_RUNG
   RUNG wire#w1
      Contact( "Unit1.Em12.ControlNodes".cmStackNgBoxLoadingUpDown.monitoring.inHomePos )
      Coil( "Unit1.Em12.ControlNodes".stackNgBox."step".transition1[340] )
   END_RUNG
   RUNG wire#w1
      Contact( "Unit1.Em12.ControlNodes".stackNgBox."step".transition1[340] )
      { S7_Templates := "time_type := Time" } #statTonTime[340].TON(pt := T#100ms, et =>)
      Move(in := #JOB_3_STEP_90, out1 => "Unit1.Em12.ControlNodes".stackNgBox.sequence.status.nextStep)
   END_RUNG
   // the same network as SCL:
   #_w1 := ("Unit1.Em12.ControlNodes".stackNgBox.sequence.status.currentStep = #JOB_3_STEP_40) AND "Unit1.Em12.ControlNodes".stackNgBox.sequence.status.seqActive;
   "Unit1.Em12.ControlNodes".stackNgBox."step".action1[340] := #_w1 AND NOT "Unit1.Em12.ControlNodes".cmStackNgBoxLoadingUpDown.monitoring.inHomePos;
   "Unit1.Em12.ControlNodes".stackNgBox."step".transition1[340] := #_w1 AND "Unit1.Em12.ControlNodes".cmStackNgBoxLoadingUpDown.monitoring.inHomePos;
   #statTonTime[340].TON(IN := #_w1 AND "Unit1.Em12.ControlNodes".stackNgBox."step".transition1[340],
                         PT := T#100ms);
   IF #statTonTime[340].Q THEN
       "Unit1.Em12.ControlNodes".stackNgBox.sequence.status.nextStep := #JOB_3_STEP_90;
   END_IF;
END_REGION

REGION Network 26: Step[390] : JOB[3] Step End
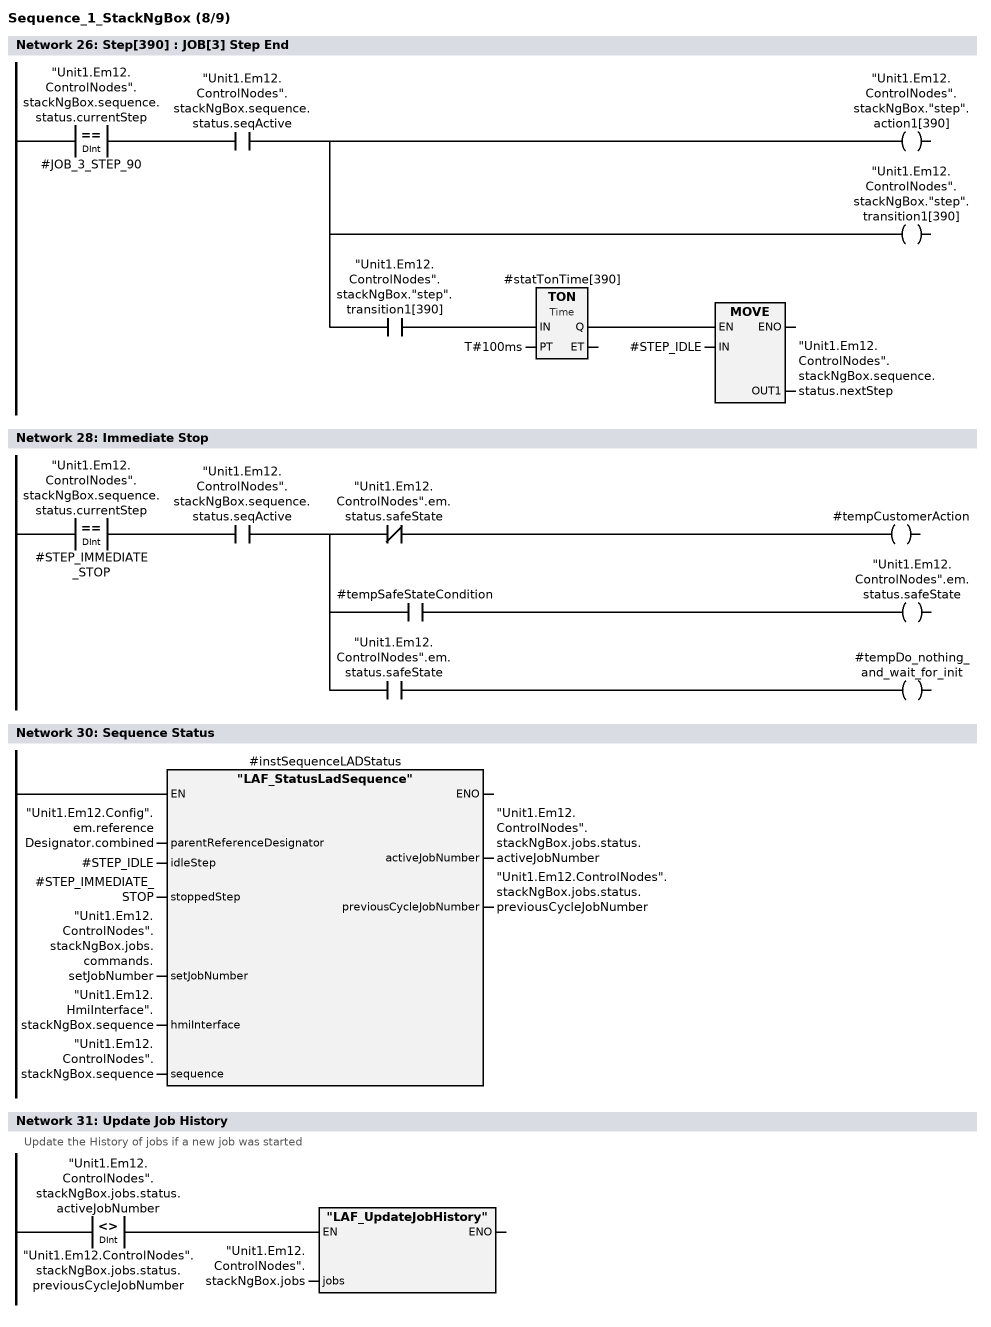
   RUNG wire#powerrail
      { S7_Templates := "SrcType := DInt" } EQ_Contact(in1 := "Unit1.Em12.ControlNodes".stackNgBox.sequence.status.currentStep, in2 := #JOB_3_STEP_90)
      Contact( "Unit1.Em12.ControlNodes".stackNgBox.sequence.status.seqActive )
      wire#w1
      Coil( "Unit1.Em12.ControlNodes".stackNgBox."step".action1[390] )
   END_RUNG
   RUNG wire#w1
      Coil( "Unit1.Em12.ControlNodes".stackNgBox."step".transition1[390] )
   END_RUNG
   RUNG wire#w1
      Contact( "Unit1.Em12.ControlNodes".stackNgBox."step".transition1[390] )
      { S7_Templates := "time_type := Time" } #statTonTime[390].TON(pt := T#100ms, et =>)
      Move(in := #STEP_IDLE, out1 => "Unit1.Em12.ControlNodes".stackNgBox.sequence.status.nextStep)
   END_RUNG
   // the same network as SCL:
   "Unit1.Em12.ControlNodes".stackNgBox."step".action1[390] := ("Unit1.Em12.ControlNodes".stackNgBox.sequence.status.currentStep = #JOB_3_STEP_90) AND "Unit1.Em12.ControlNodes".stackNgBox.sequence.status.seqActive;
   "Unit1.Em12.ControlNodes".stackNgBox."step".transition1[390] := ("Unit1.Em12.ControlNodes".stackNgBox.sequence.status.currentStep = #JOB_3_STEP_90) AND "Unit1.Em12.ControlNodes".stackNgBox.sequence.status.seqActive;
   #statTonTime[390].TON(IN := ("Unit1.Em12.ControlNodes".stackNgBox.sequence.status.currentStep = #JOB_3_STEP_90) AND "Unit1.Em12.ControlNodes".stackNgBox.sequence.status.seqActive AND "Unit1.Em12.ControlNodes".stackNgBox."step".transition1[390],
                         PT := T#100ms);
   IF #statTonTime[390].Q THEN
       "Unit1.Em12.ControlNodes".stackNgBox.sequence.status.nextStep := #STEP_IDLE;
   END_IF;
END_REGION

REGION Network 27: ******************** IMMEDIATE STOP *********************
END_REGION

REGION Network 28: Immediate Stop
   RUNG wire#powerrail
      { S7_Templates := "SrcType := DInt" } EQ_Contact(in1 := "Unit1.Em12.ControlNodes".stackNgBox.sequence.status.currentStep, in2 := #STEP_IMMEDIATE_STOP)
      Contact( "Unit1.Em12.ControlNodes".stackNgBox.sequence.status.seqActive )
      wire#w1
      I_Contact( "Unit1.Em12.ControlNodes".em.status.safeState )
      Coil( #tempCustomerAction )
   END_RUNG
   RUNG wire#w1
      Contact( #tempSafeStateCondition )
      Coil( "Unit1.Em12.ControlNodes".em.status.safeState )
   END_RUNG
   RUNG wire#w1
      Contact( "Unit1.Em12.ControlNodes".em.status.safeState )
      Coil( #tempDo_nothing_and_wait_for_init )
   END_RUNG
   // the same network as SCL:
   #_w1 := ("Unit1.Em12.ControlNodes".stackNgBox.sequence.status.currentStep = #STEP_IMMEDIATE_STOP) AND "Unit1.Em12.ControlNodes".stackNgBox.sequence.status.seqActive;
   #tempCustomerAction := #_w1 AND NOT "Unit1.Em12.ControlNodes".em.status.safeState;
   "Unit1.Em12.ControlNodes".em.status.safeState := #_w1 AND #tempSafeStateCondition;
   #tempDo_nothing_and_wait_for_init := #_w1 AND "Unit1.Em12.ControlNodes".em.status.safeState;
END_REGION

REGION Network 29: ********************** STATUS **************************
END_REGION

REGION Network 30: Sequence Status
   RUNG wire#powerrail
      #instSequenceLADStatus(parentReferenceDesignator := "Unit1.Em12.Config".em.referenceDesignator.combined, idleStep := #STEP_IDLE, stoppedStep := #STEP_IMMEDIATE_STOP, setJobNumber := "Unit1.Em12.ControlNodes".stackNgBox.jobs.commands.setJobNumber, hmiInterface := "Unit1.Em12.HmiInterface".stackNgBox.sequence, sequence := "Unit1.Em12.ControlNodes".stackNgBox.sequence, activeJobNumber => "Unit1.Em12.ControlNodes".stackNgBox.jobs.status.activeJobNumber, previousCycleJobNumber => "Unit1.Em12.ControlNodes".stackNgBox.jobs.status.previousCycleJobNumber)
   END_RUNG
   // the same network as SCL:
   #instSequenceLADStatus(parentReferenceDesignator := "Unit1.Em12.Config".em.referenceDesignator.combined,   // "LAF_StatusLadSequence"
                          idleStep := #STEP_IDLE,
                          stoppedStep := #STEP_IMMEDIATE_STOP,
                          setJobNumber := "Unit1.Em12.ControlNodes".stackNgBox.jobs.commands.setJobNumber,
                          hmiInterface := "Unit1.Em12.HmiInterface".stackNgBox.sequence,
                          sequence := "Unit1.Em12.ControlNodes".stackNgBox.sequence,
                          activeJobNumber => "Unit1.Em12.ControlNodes".stackNgBox.jobs.status.activeJobNumber,
                          previousCycleJobNumber => "Unit1.Em12.ControlNodes".stackNgBox.jobs.status.previousCycleJobNumber);
END_REGION

REGION Network 31: Update Job History
   // Update the History of jobs if a new job was started
   RUNG wire#powerrail
      { S7_Templates := "SrcType := DInt" } NE_Contact(in1 := "Unit1.Em12.ControlNodes".stackNgBox.jobs.status.activeJobNumber, in2 := "Unit1.Em12.ControlNodes".stackNgBox.jobs.status.previousCycleJobNumber)
      "LAF_UpdateJobHistory"(jobs := "Unit1.Em12.ControlNodes".stackNgBox.jobs)
   END_RUNG
   // the same network as SCL:
   IF "Unit1.Em12.ControlNodes".stackNgBox.jobs.status.activeJobNumber <> "Unit1.Em12.ControlNodes".stackNgBox.jobs.status.previousCycleJobNumber THEN
       "LAF_UpdateJobHistory"(jobs := "Unit1.Em12.ControlNodes".stackNgBox.jobs);
   END_IF;
END_REGION

REGION Network 32: Output Steps As String
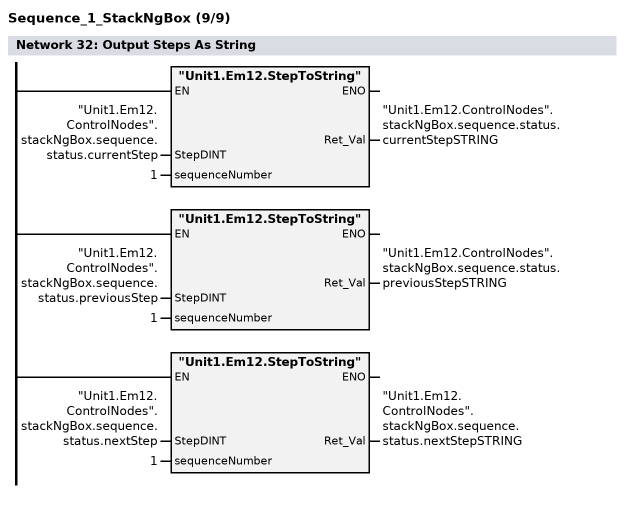
   RUNG wire#powerrail
      "Unit1.Em12.StepToString"(StepDINT := "Unit1.Em12.ControlNodes".stackNgBox.sequence.status.currentStep, sequenceNumber := 1, Ret_Val => "Unit1.Em12.ControlNodes".stackNgBox.sequence.status.currentStepSTRING)
   END_RUNG
   RUNG wire#powerrail
      "Unit1.Em12.StepToString"(StepDINT := "Unit1.Em12.ControlNodes".stackNgBox.sequence.status.previousStep, sequenceNumber := 1, Ret_Val => "Unit1.Em12.ControlNodes".stackNgBox.sequence.status.previousStepSTRING)
   END_RUNG
   RUNG wire#powerrail
      "Unit1.Em12.StepToString"(StepDINT := "Unit1.Em12.ControlNodes".stackNgBox.sequence.status.nextStep, sequenceNumber := 1, Ret_Val => "Unit1.Em12.ControlNodes".stackNgBox.sequence.status.nextStepSTRING)
   END_RUNG
   // the same network as SCL:
   "Unit1.Em12.ControlNodes".stackNgBox.sequence.status.currentStepSTRING := "Unit1.Em12.StepToString"(StepDINT := "Unit1.Em12.ControlNodes".stackNgBox.sequence.status.currentStep,
                           sequenceNumber := 1);
   "Unit1.Em12.ControlNodes".stackNgBox.sequence.status.previousStepSTRING := "Unit1.Em12.StepToString"(StepDINT := "Unit1.Em12.ControlNodes".stackNgBox.sequence.status.previousStep,
                           sequenceNumber := 1);
   "Unit1.Em12.ControlNodes".stackNgBox.sequence.status.nextStepSTRING := "Unit1.Em12.StepToString"(StepDINT := "Unit1.Em12.ControlNodes".stackNgBox.sequence.status.nextStep,
                           sequenceNumber := 1);
END_REGION
END_FUNCTION_BLOCK
